FUNCTION_BLOCK FB_CsvPersistentEventStorage IMPLEMENTS I_PersistantEventStorage
VAR
	fbFileOpen : FB_FileOpen := (sPathName := 'C:\Users\QuE\Documents\twincat_proj\Events.log', nMode := FOPEN_MODEAPPEND OR FOPEN_MODETEXT);
	fbFilePuts : FB_FilePuts;
	fbFileClose : FB_FileClose;
	eWriteState : (FILE_OPEN_TRIGGER, FILE_OPEN, WAIT_FOR_EVENT, WRITE_EVENT_TRIGGER, WRITE_EVENT, FILE_CLOSE_TRIGGER, FILE_CLOSE, ERROR);
	stEventWrittenToFile : ST_Event;
	
	CsvString : T_MaxString;
	
END_VAR

CASE eWriteState OF
	FILE_OPEN_TRIGGER : 
		fbFileOpen(bExecute := TRUE); 
		eWriteState := FILE_OPEN; 
    FILE_OPEN : 
		fbFileOpen(bExecute := FALSE); 
		IF fbFileOpen.bError THEN
			eWriteState := Error;
		ELSIF NOT fbFileOpen.bBusy AND fbFileOpen.hFile <> 0 THEN
			eWriteState := WAIT_FOR_EVENT;
		END_IF
                                          
	WAIT_FOR_EVENT :
		//Do Nothing
	
	WRITE_EVENT_TRIGGER :
		CsvString := CreateCsvString(stEvent := stEventWrittenToFile);
		fbFilePuts(bExecute := TRUE, sLine := CsvString, hFile := fbFileOpen.hFile);
		eWriteState := WRITE_EVENT;
		
	WRITE_EVENT :
		fbFilePuts(bExecute := FALSE);
		IF fbFilePuts.bError THEN
			eWriteState := Error;
		ELSIF NOT fbFilePuts.bBusy THEN
			eWriteState := FILE_CLOSE_TRIGGER;
		END_IF
	
	FILE_CLOSE_TRIGGER :
		fbFileClose(bExecute := TRUE, hFile := fbFileOpen.hFile);
		eWriteState := FILE_CLOSE;
	
	FILE_CLOSE :
		fbFileClose(bExecute := FALSE);
		IF fbFileClose.bError THEN
			eWriteState := ERROR;
		ELSIF NOT fbFileClose.bBusy THEN 
			eWriteState := FILE_OPEN_TRIGGER;
		END_IF
	
	ERROR :
		//DO NOTHING
	
END_CASE

METHOD PRIVATE CreateCsvString : T_MaxString
VAR_INPUT
	stEvent : REFERENCE TO ST_Event;
END_VAR
VAR
	TempString : T_MaxString; 
END_VAR
TempString := TO_STRING(stEvent.eEventType);
TempString :=CONCAT(STR1 := TempString, STR2 := ',');
TempString :=CONCAT(STR1 := TempString, STR2 := TO_STRING(stEvent.eEventSeverity));
TempString :=CONCAT(STR1 := TempString, STR2 := ',');
TempString :=CONCAT(STR1 := TempString, STR2 := TO_STRING(stEvent.nEventIdentity));
TempString :=CONCAT(STR1 := TempString, STR2 := ',');
TempString :=CONCAT(STR1 := TempString, STR2 := stEvent.sEventText);
TempString :=CONCAT(STR1 := TempString, STR2 := ',');
TempString :=CONCAT(STR1 := TempString, STR2 := TO_STRING(stEvent.dtTimestamp));
TempString :=CONCAT(STR1 := TempString, STR2 := '$n');

CreateCsvString := TempString;
END_METHOD

{warning 'add method implementation '}
METHOD StoreEvent : BOOL
VAR_INPUT
	stEvent	: ST_Event;
END_VAR
IF eWriteState = WAIT_FOR_EVENT THEN
	eWriteState := WRITE_EVENT_TRIGGER;
	stEventWrittenToFile := stEvent;
END_IF
END_METHOD

END_FUNCTION_BLOCK

(* stored: Version 1.1.0.1, ProductVersion 3.1.4024.12
   POU FB_CsvPersistentEventStorage: Id {03cf6f33-911d-43a9-96b4-6141ea87e407}, SpecialFunc None
   Method CreateCsvString: Id {49043991-8a88-4b26-93fc-e5eb56d6e237}
   Method StoreEvent: Id {6df6f014-49f4-4977-a877-15292f1beb46} *)
